// All OK
IF (TestInstancePathLen + TestMessageLen) <= MESSAGE_FORMATTED_STRING_MAX_NUMBER_OF_CHARACTERS THEN
    TestInstancePathProcessed := TestInstancePath;
    TestMessageProcessed := TestMessage;
// If test instance path is longer than limit, shorten it down to the allowed length minus the length of the hint '...TestName too long'. Add the hint '...TestName too long' to the test instance path. Leave no characters for the message.
ELSIF TestInstancePathLen > MESSAGE_FORMATTED_STRING_MAX_NUMBER_OF_CHARACTERS THEN
    TestInstancePathTemporary := LEFT(STR := TestInstancePath,
                                      SIZE := (MESSAGE_FORMATTED_STRING_MAX_NUMBER_OF_CHARACTERS - LEN(STR := TEST_NAME_TOO_LONG)));
    TestInstancePathProcessed := CONCAT(STR1 := TestInstancePathTemporary,
                                        STR2 := TEST_NAME_TOO_LONG);
    TestMessageProcessed := '';
// If test message is too long (so we cant fit the text "...TestMsg too long" to the end of it) , shorten it (so that we can fit the text)
ELSIF (MESSAGE_FORMATTED_STRING_MAX_NUMBER_OF_CHARACTERS - LEN(STR := TEST_MESSAGE_TOO_LONG)) >= TestInstancePathLen THEN
    TestInstancePathProcessed := TestInstancePath;
    TestMessageProcessed := LEFT(STR := TestMessage,
                                 SIZE := (MESSAGE_FORMATTED_STRING_MAX_NUMBER_OF_CHARACTERS - LEN(STR := TEST_MESSAGE_TOO_LONG) - LEN(STR := TestInstancePathProcessed)));
    TestMessageProcessed := CONCAT(STR1 := TestMessageProcessed,
                                   STR2 := TEST_MESSAGE_TOO_LONG);
// If test instance path is too long (length is between 233 and 252 characters long), shorten it and add the text '...TestName too long'. Leave no characters for the message
ELSE
    TestInstancePathTemporary := LEFT(STR := TestInstancePath,
                                      SIZE := (MESSAGE_FORMATTED_STRING_MAX_NUMBER_OF_CHARACTERS - LEN(STR := TEST_NAME_TOO_LONG)));
    TestInstancePathProcessed := CONCAT(STR1 := TestInstancePathTemporary,
                                        STR2 := TEST_NAME_TOO_LONG);
    TestMessageProcessed := '';
END_IF

END_FUNCTION_BLOCK

// ---- POUs/Functions/F_AnyTypeClassToString.TcPOU
// This function takes the type-class of a ANY-variable and returns the STRING representation of it.
FUNCTION F_AnyTypeClassToString : STRING
VAR_INPUT
    AnyTypeClass : __SYSTEM.TYPE_CLASS;
END_VAR

CASE UDINT_TO_INT(AnyTypeClass) OF
    IBaseLibrary.TypeClass.TYPE_BOOL :
        F_AnyTypeClassToString := 'BOOL';

    IBaseLibrary.TypeClass.TYPE_BIT :
        F_AnyTypeClassToString := 'BIT';

    IBaseLibrary.TypeClass.TYPE_BYTE :
        F_AnyTypeClassToString := 'BYTE';

    IBaseLibrary.TypeClass.TYPE_WORD :
        F_AnyTypeClassToString := 'WORD';

    IBaseLibrary.TypeClass.TYPE_DWORD :
        F_AnyTypeClassToString := 'DWORD';

    IBaseLibrary.TypeClass.TYPE_LWORD :
        F_AnyTypeClassToString := 'LWORD';

    IBaseLibrary.TypeClass.TYPE_SINT :
        F_AnyTypeClassToString := 'SINT';

    IBaseLibrary.TypeClass.TYPE_INT :
        F_AnyTypeClassToString := 'INT';

    IBaseLibrary.TypeClass.TYPE_DINT :
        F_AnyTypeClassToString := 'DINT';

    IBaseLibrary.TypeClass.TYPE_LINT :
        F_AnyTypeClassToString := 'LINT';

    IBaseLibrary.TypeClass.TYPE_USINT :
        F_AnyTypeClassToString := 'USINT';

    IBaseLibrary.TypeClass.TYPE_UINT :
        F_AnyTypeClassToString := 'UINT';

    IBaseLibrary.TypeClass.TYPE_UDINT :
        F_AnyTypeClassToString := 'UDINT';

    IBaseLibrary.TypeClass.TYPE_ULINT :
        F_AnyTypeClassToString := 'ULINT';

    IBaseLibrary.TypeClass.TYPE_REAL :
        F_AnyTypeClassToString := 'REAL';

    IBaseLibrary.TypeClass.TYPE_LREAL :
        F_AnyTypeClassToString := 'LREAL';

    IBaseLibrary.TypeClass.TYPE_STRING :
        F_AnyTypeClassToString := 'STRING';

    IBaseLibrary.TypeClass.TYPE_WSTRING :
        F_AnyTypeClassToString := 'WSTRING';

    IBaseLibrary.TypeClass.TYPE_TIME :
        F_AnyTypeClassToString := 'TIME';

    IBaseLibrary.TypeClass.TYPE_DATE :
        F_AnyTypeClassToString := 'DATE';

    IBaseLibrary.TypeClass.TYPE_DATEANDTIME :
        F_AnyTypeClassToString := 'DATEANDTIME';

    IBaseLibrary.TypeClass.TYPE_TIMEOFDAY :
        F_AnyTypeClassToString := 'TIMEOFDAY';

    IBaseLibrary.TypeClass.TYPE_POINTER :
        F_AnyTypeClassToString := 'POINTER';

    IBaseLibrary.TypeClass.TYPE_REFERENCE :
        F_AnyTypeClassToString := 'REFERENCE';

    IBaseLibrary.TypeClass.TYPE_SUBRANGE :
        F_AnyTypeClassToString := 'SUBRANGE';

    IBaseLibrary.TypeClass.TYPE_ENUM :
        F_AnyTypeClassToString := 'ENUM';

    IBaseLibrary.TypeClass.TYPE_ARRAY :
        F_AnyTypeClassToString := 'ARRAY';

    IBaseLibrary.TypeClass.TYPE_PARAMS :
        F_AnyTypeClassToString := 'PARAMS';

    IBaseLibrary.TypeClass.TYPE_USERDEF :
        F_AnyTypeClassToString := 'USERDEF';

    IBaseLibrary.TypeClass.TYPE_NONE :
        F_AnyTypeClassToString := 'NONE';

    IBaseLibrary.TypeClass.TYPE_ANY :
        F_AnyTypeClassToString := 'ANY';

    IBaseLibrary.TypeClass.TYPE_ANYBIT :
        F_AnyTypeClassToString := 'ANYBIT';

    IBaseLibrary.TypeClass.TYPE_ANYDATE :
        F_AnyTypeClassToString := 'ANYDATE';

    IBaseLibrary.TypeClass.TYPE_ANYINT :
        F_AnyTypeClassToString := 'ANYINT';

    IBaseLibrary.TypeClass.TYPE_ANYNUM :
        F_AnyTypeClassToString := 'ANYNUM';

    IBaseLibrary.TypeClass.TYPE_ANYREAL :
        F_AnyTypeClassToString := 'ANYREAL';

    IBaseLibrary.TypeClass.TYPE_LAZY :
        F_AnyTypeClassToString := 'LAZY';

    IBaseLibrary.TypeClass.TYPE_LTIME :
        F_AnyTypeClassToString := 'LTIME';

    IBaseLibrary.TypeClass.TYPE_BITCONST :
        F_AnyTypeClassToString := 'BITCONST';

    IBaseLibrary.TypeClass.TYPE_INTERFACE :
        F_AnyTypeClassToString := 'INTERFACE';

    ELSE
        F_AnyTypeClassToString := 'UNKNOWN';

END_CASE

END_FUNCTION

// ---- POUs/Functions/RUN.TcPOU
(*
    This function runs all test suites that have been initialized.
    The test suites are run in parallel (all at once).
*)
FUNCTION RUN

GVL_TcUnit.TcUnitRunner.RunTestSuiteTests();

END_FUNCTION

// ---- POUs/Functions/TEST_ORDERED.TcPOU
(* This function declares a new ordered test (if it has not been already declared in an earlier cycle).
   The test declared by this function will run in the order it is called, so if we have two tests:
   TEST_ORDERED('Test_1')
   TEST_ORDERED('Test_2')
   All asserts of Test_2 will be ignored until Test_1 is declared with TEST_FINISHED().

   The function returns TRUE if it's time to run this test (and thus asserts can be made)
   The function returns FALSE if it's not time to run this test (because a previous test has not been finished)
   If the function returns FALSE (and it's thus not time to run the test), any eventual asserts done for this 
   test will be ignored. It thus makes sense to call this function in a manner like:
   
    IF TEST_ORDERED('Testname') THEN
        fbFunctionBlockUnderTest();
        
        AssertEquals(Expected := 'SomeValue',
                     Actual := fbFunctionBlockUnderTest.Out,
                     Message := 'Test failed');
        TEST_FINISHED();
    END_IF

*)
FUNCTION TEST_ORDERED : BOOL
VAR_INPUT
    TestName : T_MaxString;
END_VAR
VAR
    CounterTestSuiteAddress : UINT;
    Test : REFERENCE TO FB_Test;
END_VAR

TestName := F_LTrim(in := F_RTrim(in := TestName));

// Mark this test as the current one being executed
GVL_TcUnit.CurrentTestNameBeingCalled := TestName;

(* Check if combination of address for the test suite and test name already exists.
   For every test suite the name of the test case needs to be unique.
   If a test with this name already exists, don't add it to the available tests.
   Otherwise, add it to the available tests *)

FOR CounterTestSuiteAddress := 1 TO GVL_TcUnit.NumberOfInitializedTestSuites BY 1 DO

    // Look for the test suite by comparing to the one that is currently running
    IF GVL_TcUnit.TestSuiteAddresses[CounterTestSuiteAddress] = GVL_TcUnit.CurrentTestSuiteBeingCalled THEN
        Test REF= GVL_TcUnit.TestSuiteAddresses[CounterTestSuiteAddress]^.AddTest(TestName := TestName, IsTestOrdered := TRUE);
        GVL_TcUnit.CurrentTestIsFinished := GVL_TcUnit.TestSuiteAddresses[CounterTestSuiteAddress]^.IsTestFinished(TestName := TestName);

        // Check that no previous code has set the currently running test to ignored (for example by setting the test to DISABLED
        IF NOT GVL_TcUnit.IgnoreCurrentTest THEN
            (* If the current test is not the current in the sequence of tests, set it to ignored until it is its turn to run
               If the current test is the one supposed to be run, check whether it has finished running or not *)
            IF GVL_TcUnit.TestSuiteAddresses[CounterTestSuiteAddress]^.GetTestOrderNumber(TestName := TestName) =
                GVL_TcUnit.CurrentlyRunningOrderedTestInTestSuite[CounterTestSuiteAddress] THEN
                // Check if test if finished, if so, increase the order number of this test suite to the next test
                IF GVL_TcUnit.CurrentTestIsFinished THEN
                    GVL_TcUnit.CurrentlyRunningOrderedTestInTestSuite[CounterTestSuiteAddress] := GVL_TcUnit.CurrentlyRunningOrderedTestInTestSuite[CounterTestSuiteAddress] + 1;
                    // No need to execute the test if it is already finished
                    TEST_ORDERED := FALSE;
                    GVL_TcUnit.IgnoreCurrentTest := TRUE;
                ELSE
                    // Start or continue executing test
                    IF __ISVALIDREF(Test) THEN
                        Test.SetStartedAtIfNotSet(Timestamp := F_GetCpuCounterAs64bit(GVL_TcUnit.GetCpuCounter));
                    END_IF
                    TEST_ORDERED := TRUE;
                END_IF
            ELSE
                // If this is not the current test that we are supposed to run, ignore it until it is its turn
                TEST_ORDERED := FALSE;
                GVL_TcUnit.IgnoreCurrentTest := TRUE;
			END_IF
        // This test should be ignored
        ELSE
            TEST_ORDERED := FALSE;
            GVL_TcUnit.IgnoreCurrentTest := TRUE;
		END_IF
        RETURN;
    END_IF
END_FOR

END_FUNCTION

// ---- POUs/FB_AdsLogStringMessageFifoQueue.TcPOU
(* This function block is responsible for making sure that the ADSLOGSTR-messages to the ADS-router are transmitted
   cyclically and not in a burst. The reason this is necessary is because that if too many messages are sent at the
   same time some get lost and are never printed to the error list output
*)
FUNCTION_BLOCK FB_AdsLogStringMessageFifoQueue
VAR
    ArrayBuffer : ARRAY[0..((GVL_Param_TcUnit.AdsLogMessageFifoRingBufferSize * (SIZEOF(ST_ADSLogStringMessage) + MEM_RING_BUFFER_INTERNAL_USE_PER_DATA_RECORD)) - 1)] OF BYTE;
    MemRingBuffer : FB_MemRingBuffer;
    TimerBetweenMessages : TON := (IN := TRUE, PT := TIME_BETWEEN_MESSAGES);
END_VAR
VAR CONSTANT
    MEM_RING_BUFFER_INTERNAL_USE_PER_DATA_RECORD : USINT := 4;
    TIME_BETWEEN_MESSAGES : TIME := T#10MS;
END_VAR
VAR_TEMP
    MessageToBeSent : ST_AdsLogStringMessage;
    ErrorGet : BOOL;
    ReturnValue : DINT;
END_VAR

TimerBetweenMessages();
IF GetLogCount() > 0 THEN
    // Timer has elapsed, print message
    IF TimerBetweenMessages.Q THEN
        GetAndRemoveLogFromQueue(AdsLogStringMessage => MessageToBeSent,
                                 Error => ErrorGet);
        IF NOT ErrorGet THEN
            ReturnValue := ADSLOGSTR(msgCtrlMask := MessageToBeSent.MsgCtrlMask,
                                     msgFmtStr := MessageToBeSent.MsgFmtStr,
                                     strArg := MessageToBeSent.StrArg);
        END_IF
        TimerBetweenMessages(IN := FALSE); // Reset timer
        TimerBetweenMessages.IN := TRUE;
    END_IF
END_IF

(* Reads and removes the oldest message *)
METHOD PRIVATE GetAndRemoveLogFromQueue
VAR_OUTPUT
    AdsLogStringMessage : ST_ADSLogStringMessage;
    Error : BOOL; // Buffer empty
END_VAR
MemRingBuffer.A_RemoveHead(pRead := ADR(AdsLogStringMessage),
                           cbRead := SIZEOF(ST_ADSLogStringMessage),
                           pBuffer := ADR(ArrayBuffer),
                           cbBuffer := SIZEOF(ArrayBuffer));
Error := NOT MemRingBuffer.bOk;
END_METHOD

METHOD PRIVATE GetLogCount : UDINT
GetLogCount := MemRingBuffer.nCount;
END_METHOD

// Writes a new data set into the ring buffer
METHOD INTERNAL WriteLog
VAR_INPUT
    MsgCtrlMask : DWORD;
    MsgFmtStr : T_MaxString;
    StrArg : T_MaxString;
END_VAR
VAR_OUTPUT
    Error : BOOL; // Buffer overflow
END_VAR
VAR
    AdsLogStringMessage : ST_AdsLogStringMessage;
END_VAR
// Only log message types of ERROR if log extended results is not enabled
IF GVL_Param_TcUnit.AdsLoggerEnablePublish AND_THEN (MsgCtrlMask = ADSLOG_MSGTYPE_ERROR OR GVL_Param_TcUnit.LogExtendedResults) THEN
    AdsLogStringMessage.MsgCtrlMask := MsgCtrlMask;
    AdsLogStringMessage.MsgFmtStr := MsgFmtStr;
    AdsLogStringMessage.StrArg := StrArg;

    MemRingBuffer.A_AddTail(pWrite := ADR(AdsLogStringMessage),
                            cbWrite := SIZEOF(ST_AdsLogStringMessage),
                            pBuffer := ADR(ArrayBuffer),
                            cbBuffer := SIZEOF(ArrayBuffer));

    Error := NOT MemRingBuffer.bOk;
END_IF
END_METHOD

END_FUNCTION_BLOCK

// ---- POUs/FB_FileControl.TcPOU
// This functionblock can open, close, read, write and delete files on the local filesystem
FUNCTION_BLOCK FB_FileControl
VAR
    FileAccessMode : SysFile.ACCESS_MODE := SysFile.AM_APPEND_PLUS; // Append_Plus creates the file if it doesn't exist yet. 
    FileHandle : SysFile.SysTypes.RTS_IEC_HANDLE;
END_VAR

// Closes the currently opened file.
METHOD PUBLIC Close : SysFile.SysTypes.RTS_IEC_RESULT;
IF FileHandle <> SysFile.SysTypes.RTS_INVALID_HANDLE THEN
    Close := SysFile.SysFileClose(hFile := FileHandle);
ELSE
    Close := SysDir.CmpErrors.Errors.ERR_INVALID_HANDLE;
END_IF
END_METHOD

// Deletes a file specified by name, if it exists.
METHOD PUBLIC Delete : SysFile.SysTypes.RTS_IEC_RESULT;
VAR_INPUT
    // File name can contain an absolute or relative path to the file. Path entries must be separated with a forward slash (/)
    FileName : T_MaxString;
END_VAR
Delete := SysFile.SysFileDelete(szFileName := FileName);
END_METHOD

// Opens a file
METHOD PUBLIC Open : SysFile.SysTypes.RTS_IEC_RESULT;
VAR_INPUT
    FileName : T_MaxString := 'filepath/output.xml';  // File name can contain an absolute or relative path to the file. Path entries must be separated with a Slash (/)
    FileAccessMode : SysFile.ACCESS_MODE := SysFile.ACCESS_MODE.AM_APPEND_PLUS;
END_VAR
FileHandle := SysFile.SysFileOpen(szFile := Filename,
                                  am := FileAccessMode,
                                  pResult := ADR(Open));
END_METHOD

// Reads a file from disk into the buffer
METHOD PUBLIC Read : SysFile.SysTypes.RTS_IEC_RESULT;
VAR_INPUT
    BufferPointer : POINTER TO BYTE; // Call with ADR();
    Size : UDINT; // Call with SIZEOF(); 
END_VAR
VAR_OUTPUT
    FileSize : SysFile.SysTypes.RTS_IEC_SIZE;
END_VAR
IF FileHandle <> SysFile.SysTypes.RTS_INVALID_HANDLE THEN
    FileSize := SysFile.SysFileRead(hFile := FileHandle, 
                                    pbyBuffer := BufferPointer,
                                    ulSize := Size,
                                    pResult := ADR(Read));
ELSE
    Read := SysDir.CmpErrors.Errors.ERR_INVALID_HANDLE;
END_IF
END_METHOD

// Writes the contents of the buffer into a file.
METHOD PUBLIC Write : SysFile.SysTypes.RTS_IEC_RESULT;
VAR_INPUT
    BufferPointer : POINTER TO BYTE; // Call with ADR();
    Size : UDINT; // Call with SIZEOF();
END_VAR
IF FileHandle <> SysFile.SysTypes.RTS_INVALID_HANDLE THEN
    SysFile.SysFileWrite(hFile := FileHandle,
                         pbyBuffer := BufferPointer,
                         ulSize := Size,
                         pResult := ADR(Write));
ELSE
    Write := SysDir.CmpErrors.Errors.ERR_INVALID_HANDLE;
END_IF
END_METHOD

END_FUNCTION_BLOCK

// ---- POUs/Functions/IS_TEST_FINISHED.TcPOU
// Check if a certain test in the current suite is finished
FUNCTION IS_TEST_FINISHED : BOOL
VAR_INPUT
    TestName : T_MaxString;
END_VAR
VAR
    Counter : UINT;
    CurrentTest : FB_Test;
END_VAR

TestName := F_LTrim(in := F_RTrim(in := TestName));

IS_TEST_FINISHED := FALSE;

FOR Counter := 1 TO GVL_TcUnit.CurrentTestSuiteBeingCalled^.GetNumberOfTests() BY 1 DO
    CurrentTest := GVL_TcUnit.CurrentTestSuiteBeingCalled^.Tests[Counter];
    IF CurrentTest.TestName = TestName THEN
        IS_TEST_FINISHED := CurrentTest.IsFinished();
        RETURN;
    END_IF
END_FOR

END_FUNCTION

// ---- POUs/Functions/TCUNIT_ADSLOGSTR.TcPOU
(* This function allows to put ADS strings into the TcUnit ADS message buffer. If ADSLOGSTR() is used directly,
   the messages can come out of sequence in relation to the message created by TcUnit as TcUnit buffers the messages to
   not overflow the ADS message router. By using this function, the ADS-messages are put in the same buffer as
   TcUnit is using for its output and thus the sequence will be correct *)
FUNCTION TCUNIT_ADSLOGSTR
VAR_INPUT
    msgCtrlMask : DWORD; // Message control mask
    msgFmtStr : T_MaxString; // Message format string
    strArg : T_MaxString; // STRING argument
END_VAR

GVL_TcUnit.AdsMessageQueue.WriteLog(MsgCtrlMask := msgCtrlMask,
                                    MsgFmtStr := msgFmtStr,
                                    StrArg := strArg);

END_FUNCTION

// ---- POUs/Functions/TEST_FINISHED.TcPOU
// Sets the currently running test as finished
FUNCTION TEST_FINISHED : BOOL
VAR
    TestName : T_MaxString;
    Counter : UINT := 0;
    FinishedAt : LWORD;
END_VAR

// Get the timestamp directly when the test has finished
FinishedAt := F_GetCpuCounterAs64bit(GVL_TcUnit.GetCpuCounter);

// Grab the currently running test name
TestName := GVL_TcUnit.CurrentTestNameBeingCalled;

TEST_FINISHED := FALSE;
(* Find the test suite and:
   1. Set the test in that test suite as finished
   2. Calculate and set the number of asserts made for that test
*)
FOR Counter := 1 TO GVL_TcUnit.NumberOfInitializedTestSuites BY 1 DO
    IF GVL_TcUnit.TestSuiteAddresses[Counter] = GVL_TcUnit.CurrentTestSuiteBeingCalled THEN
        GVL_TcUnit.TestSuiteAddresses[Counter]^.SetTestFinished(TestName := GVL_TcUnit.CurrentTestNameBeingCalled, FinishedAt := FinishedAt);
        GVL_TcUnit.TestSuiteAddresses[Counter]^.CalculateAndSetNumberOfAssertsForTest(TestName := GVL_TcUnit.CurrentTestNameBeingCalled);
        GVL_TcUnit.CurrentTestIsFinished := TRUE;
        TEST_FINISHED := TRUE;
        RETURN;
    END_IF
END_FOR

END_FUNCTION

// ---- POUs/Functions/TEST_FINISHED_NAMED.TcPOU
(* Sets a test defined by TestName as finished. Note that the TestName-input must match
   a TestName that has been previously defined in this test suite. *)
FUNCTION TEST_FINISHED_NAMED
VAR_INPUT
    TestName : T_MaxString;
END_VAR
VAR
    Counter : UINT := 0;
    FoundTestName : BOOL := FALSE;
    FinishedAt : LWORD; // cpu cycle counter in 100ns precision
END_VAR
VAR_STAT
    FailedLookupCounter : UINT := 0;
    AlreadyPrintedFinalWarning : BOOL := FALSE;
END_VAR
VAR CONSTANT
    MaxNumberOfNonExistentTestNamesFailedLookups : UINT := 3;
END_VAR

TestName := F_LTrim(in := F_RTrim(in := TestName));
FinishedAt := F_GetCpuCounterAs64bit(GVL_TcUnit.GetCpuCounter);

(* Find the test suite and:
   1. Set the test in that test suite as finished
   2. Calculate and set the number of asserts made for that test
*)
FOR Counter := 1 TO GVL_TcUnit.NumberOfInitializedTestSuites BY 1 DO
    IF GVL_TcUnit.TestSuiteAddresses[Counter] = GVL_TcUnit.CurrentTestSuiteBeingCalled THEN
        FoundTestName := GVL_TcUnit.TestSuiteAddresses[Counter]^.SetTestFinished(TestName := TestName, FinishedAt := FinishedAt);
        IF NOT FoundTestName THEN
            IF FailedLookupCounter < MaxNumberOfNonExistentTestNamesFailedLookups THEN
                GVL_TcUnit.AdsMessageQueue.WriteLog(MsgCtrlMask := ADSLOG_MSGTYPE_ERROR,
                                                    MsgFmtStr := 'Failed to find test $'%s$'',
                                                    StrArg := TestName);
                FailedLookupCounter := FailedLookupCounter + 1;
                (* Abort TcUnit *)
                GVL_TcUnit.TcUnitRunner.AbortRunningTestSuiteTests();
            ELSIF NOT AlreadyPrintedFinalWarning THEN
                GVL_TcUnit.AdsMessageQueue.WriteLog(MsgCtrlMask := ADSLOG_MSGTYPE_ERROR,
                                                    MsgFmtStr := 'Excess failed attempts to mark test finished, failed. Further warnings will be suppressed',
                                                    StrArg := TestName);
                AlreadyPrintedFinalWarning := TRUE;
            END_IF
        ELSE
            GVL_TcUnit.TestSuiteAddresses[Counter]^.CalculateAndSetNumberOfAssertsForTest(TestName := TestName);
            GVL_TcUnit.CurrentTestIsFinished := TRUE;
        END_IF
        RETURN;
    END_IF
END_FOR

END_FUNCTION

// ---- POUs/Functions/WRITE_PROTECTED_/WRITE_PROTECTED_BOOL.TcPOU
FUNCTION WRITE_PROTECTED_BOOL
VAR_INPUT
    Ptr : POINTER TO BOOL;
    Value : BOOL;
END_VAR

Ptr^ := Value;

END_FUNCTION

// ---- POUs/Functions/WRITE_PROTECTED_/WRITE_PROTECTED_BYTE.TcPOU
FUNCTION WRITE_PROTECTED_BYTE
VAR_INPUT
    Ptr : POINTER TO BYTE;
    Value : BYTE;
END_VAR

Ptr^ := Value;

END_FUNCTION

// ---- POUs/Functions/WRITE_PROTECTED_/WRITE_PROTECTED_DATE.TcPOU
FUNCTION WRITE_PROTECTED_DATE
VAR_INPUT
    Ptr : POINTER TO DATE;
    Value : DATE;
END_VAR

Ptr^ := Value;

END_FUNCTION

// ---- POUs/Functions/WRITE_PROTECTED_/WRITE_PROTECTED_DATE_AND_TIME.TcPOU
FUNCTION WRITE_PROTECTED_DATE_AND_TIME
VAR_INPUT
    Ptr : POINTER TO DATE_AND_TIME;
    Value : DATE_AND_TIME;
END_VAR

Ptr^ := Value;

END_FUNCTION

// ---- POUs/Functions/WRITE_PROTECTED_/WRITE_PROTECTED_DINT.TcPOU
FUNCTION WRITE_PROTECTED_DINT
VAR_INPUT
    Ptr : POINTER TO DINT;
    Value : DINT;
END_VAR

Ptr^ := Value;

END_FUNCTION

// ---- POUs/Functions/WRITE_PROTECTED_/WRITE_PROTECTED_DWORD.TcPOU
FUNCTION WRITE_PROTECTED_DWORD
VAR_INPUT
    Ptr : POINTER TO DWORD;
    Value : DWORD;
END_VAR

Ptr^ := Value;

END_FUNCTION

// ---- POUs/Functions/WRITE_PROTECTED_/WRITE_PROTECTED_INT.TcPOU
FUNCTION WRITE_PROTECTED_INT
VAR_INPUT
    Ptr : POINTER TO INT;
    Value : INT;
END_VAR

Ptr^ := Value;

END_FUNCTION

// ---- POUs/Functions/WRITE_PROTECTED_/WRITE_PROTECTED_LREAL.TcPOU
FUNCTION WRITE_PROTECTED_LREAL
VAR_INPUT
    Ptr : POINTER TO LREAL;
    Value : LREAL;
END_VAR

Ptr^ := Value;

END_FUNCTION

// ---- POUs/Functions/WRITE_PROTECTED_/WRITE_PROTECTED_REAL.TcPOU
FUNCTION WRITE_PROTECTED_REAL
VAR_INPUT
    Ptr : POINTER TO REAL;
    Value : REAL;
END_VAR

Ptr^ := Value;

END_FUNCTION

// ---- POUs/Functions/WRITE_PROTECTED_/WRITE_PROTECTED_SINT.TcPOU
FUNCTION WRITE_PROTECTED_SINT
VAR_INPUT
    Ptr : POINTER TO SINT;
    Value : SINT;
END_VAR

Ptr^ := Value;

END_FUNCTION

// ---- POUs/Functions/WRITE_PROTECTED_/WRITE_PROTECTED_STRING.TcPOU
FUNCTION WRITE_PROTECTED_STRING
VAR_INPUT
    Ptr : POINTER TO STRING;
    Value : STRING;
END_VAR

Ptr^ := Value;

END_FUNCTION

// ---- POUs/Functions/WRITE_PROTECTED_/WRITE_PROTECTED_WSTRING.TcPOU
FUNCTION WRITE_PROTECTED_WSTRING
VAR_INPUT
    Ptr : POINTER TO WSTRING;
    Value : WSTRING;
END_VAR

Ptr^ := Value;

END_FUNCTION

// ---- POUs/Functions/WRITE_PROTECTED_/WRITE_PROTECTED_TIME.TcPOU
FUNCTION WRITE_PROTECTED_TIME
VAR_INPUT
    Ptr : POINTER TO TIME;
    Value : TIME;
END_VAR

Ptr^ := Value;

END_FUNCTION

// ---- POUs/Functions/WRITE_PROTECTED_/WRITE_PROTECTED_TIME_OF_DAY.TcPOU
FUNCTION WRITE_PROTECTED_TIME_OF_DAY
VAR_INPUT
    Ptr : POINTER TO TIME_OF_DAY;
    Value : TIME_OF_DAY;
END_VAR

Ptr^ := Value;

END_FUNCTION

// ---- POUs/Functions/WRITE_PROTECTED_/WRITE_PROTECTED_UDINT.TcPOU
FUNCTION WRITE_PROTECTED_UDINT
VAR_INPUT
    Ptr : POINTER TO UDINT;
    Value : UDINT;
END_VAR

Ptr^ := Value;

END_FUNCTION

// ---- POUs/Functions/WRITE_PROTECTED_/WRITE_PROTECTED_UINT.TcPOU
FUNCTION WRITE_PROTECTED_UINT
VAR_INPUT
    Ptr : POINTER TO UINT;
    Value : UINT;
END_VAR

Ptr^ := Value;

END_FUNCTION

// ---- POUs/Functions/WRITE_PROTECTED_/WRITE_PROTECTED_ULINT.TcPOU
FUNCTION WRITE_PROTECTED_ULINT
VAR_INPUT
    Ptr : POINTER TO ULINT;
    Value : ULINT;
END_VAR

Ptr^ := Value;

END_FUNCTION

// ---- POUs/Functions/WRITE_PROTECTED_/WRITE_PROTECTED_LWORD.TcPOU
FUNCTION WRITE_PROTECTED_LWORD
VAR_INPUT
    Ptr : POINTER TO LWORD;
    Value : LWORD;
END_VAR

Ptr^ := Value;

END_FUNCTION

// ---- POUs/Functions/WRITE_PROTECTED_/WRITE_PROTECTED_LINT.TcPOU
FUNCTION WRITE_PROTECTED_LINT
VAR_INPUT
    Ptr : POINTER TO LINT;
    Value : LINT;
END_VAR

Ptr^ := Value;

END_FUNCTION

// ---- POUs/Functions/WRITE_PROTECTED_/WRITE_PROTECTED_USINT.TcPOU
FUNCTION WRITE_PROTECTED_USINT
VAR_INPUT
    Ptr : POINTER TO USINT;
    Value : USINT;
END_VAR

Ptr^ := Value;

END_FUNCTION

// ---- POUs/Functions/WRITE_PROTECTED_/WRITE_PROTECTED_WORD.TcPOU
FUNCTION WRITE_PROTECTED_WORD
VAR_INPUT
    Ptr : POINTER TO WORD;
    Value : WORD;
END_VAR

Ptr^ := Value;

END_FUNCTION
